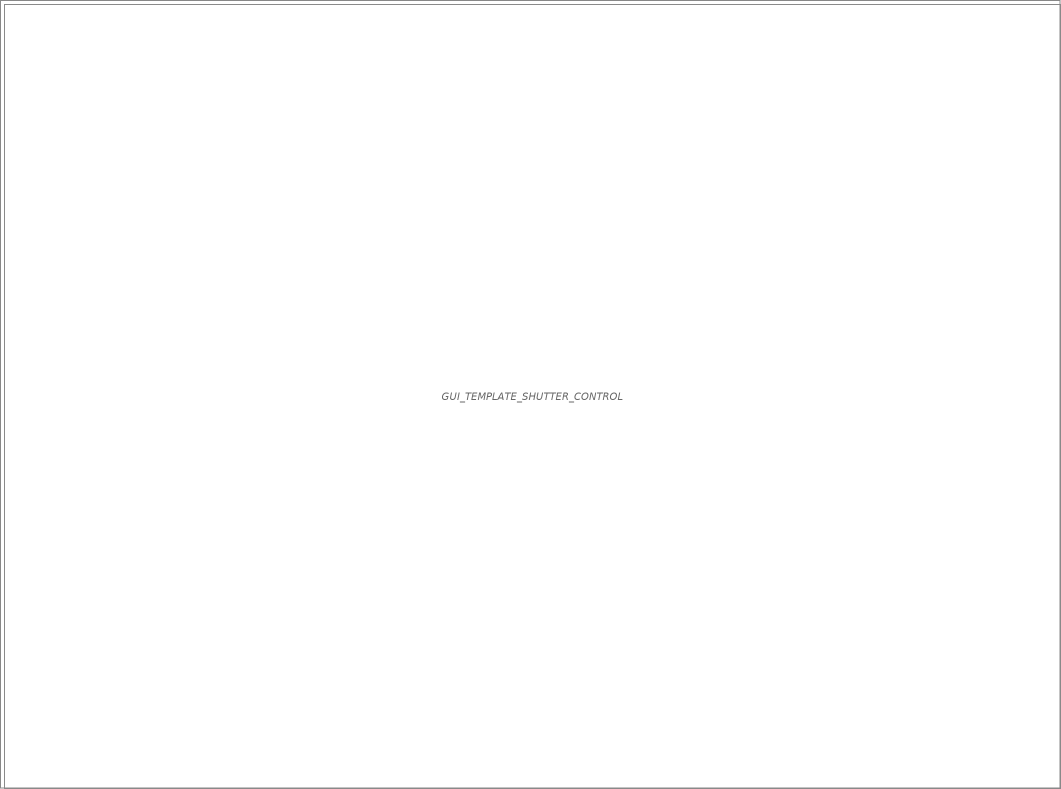
VISUALIZATION GUI_TEMPLATE_NOTT_SHUTTER  // 1061x789
VAR_IN_OUT
	m_Instance:	FB_NOTT_MOTOR;
END_VAR
    TabControl (4,4 1057x785)
        shows GUI_TEMPLATE_SHUTTER_CONTROL(m_Instance := m_Instance)
        shows GUI_TEMPLATE_NOTT_MOTOR_CONFIG(m_Instance := m_Instance)
        [0]: TabTitle=Shutter Control
        [1]: TabTitle=Config
END_VISUALIZATION

(* stored: Version 1.1.0.1, ProductVersion 3.1.4024.14
   Visu GUI_TEMPLATE_NOTT_SHUTTER: Id {8badbb78-d0c8-45d7-a743-dc07c9b258ee} *)
